(* IEC 61131-3 sources: MSMP/PLC_Station/Source/Programs, 5 files *)

(* ---- PRG_CANopen.st ---- *)
PROGRAM PRG_CANopen
VAR
 CanMgr:FB_CANopenManager;
END_VAR
CanMgr(Enable:=TRUE);
// TODO: Read 6 CANopen encoders

(* ---- PRG_Diagnostics.st ---- *)
PROGRAM PRG_Diagnostics
VAR
 Diag:FB_Diagnostics;
END_VAR
Diag(CAN_OK:=TRUE,MODBUS_OK:=TRUE);

(* ---- PRG_Main.st ---- *)
PROGRAM PRG_Main
VAR
    System : FB_System;
END_VAR

System(Enable:=TRUE);

// TODO:
// Read CANopen
// Update gStation
// Update Modbus Registers

(* ---- PRG_Modbus.st ---- *)
PROGRAM PRG_Modbus
VAR
 MB:FB_ModbusSlave;
 MAP:FB_ModbusMapping;
END_VAR
MB(Enable:=TRUE);
MAP(Enable:=TRUE);

(* ---- PRG_Station.st ---- *)
PROGRAM PRG_Station

VAR
    Acquire : FB_DataAcquisition;
    EncMgr  : FB_EncoderManager;
    StaMgr  : FB_StationManager;
END_VAR

Acquire(Enable:=TRUE);
EncMgr(Enable:=TRUE);
StaMgr(Enable:=TRUE);
